// Mitsubishi GX Works2 project: 기말   PLC: Q02/Q02H

PROGRAM MAIN
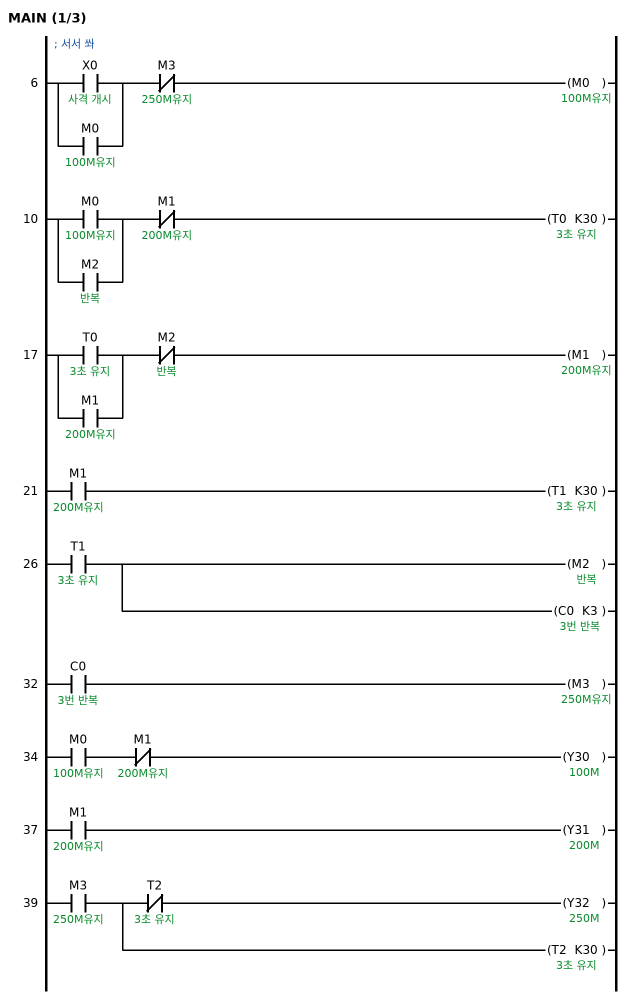
; 서서 쏴
6     LD      X0  ; 사격 개시
      OR      M0  ; 100M유지
      ANI     M3  ; 250M유지
      OUT     M0  ; 100M유지
10    LD      M0  ; 100M유지
      OR      M2  ; 반복
      ANI     M1  ; 200M유지
      OUT     T0 K30  ; 3초 유지
17    LD      T0  ; 3초 유지
      OR      M1  ; 200M유지
      ANI     M2  ; 반복
      OUT     M1  ; 200M유지
21    LD      M1  ; 200M유지
      OUT     T1 K30  ; 3초 유지
26    LD      T1  ; 3초 유지
      OUT     M2  ; 반복
      OUT     C0 K3  ; 3번 반복
32    LD      C0  ; 3번 반복
      OUT     M3  ; 250M유지
34    LD      M0  ; 100M유지
      ANI     M1  ; 200M유지
      OUT     Y30  ; 100M
37    LD      M1  ; 200M유지
      OUT     Y31  ; 200M
39    LD      M3  ; 250M유지
      MPS
      ANI     T2  ; 3초 유지
      OUT     Y32  ; 250M
      MPP
      OUT     T2 K30  ; 3초 유지
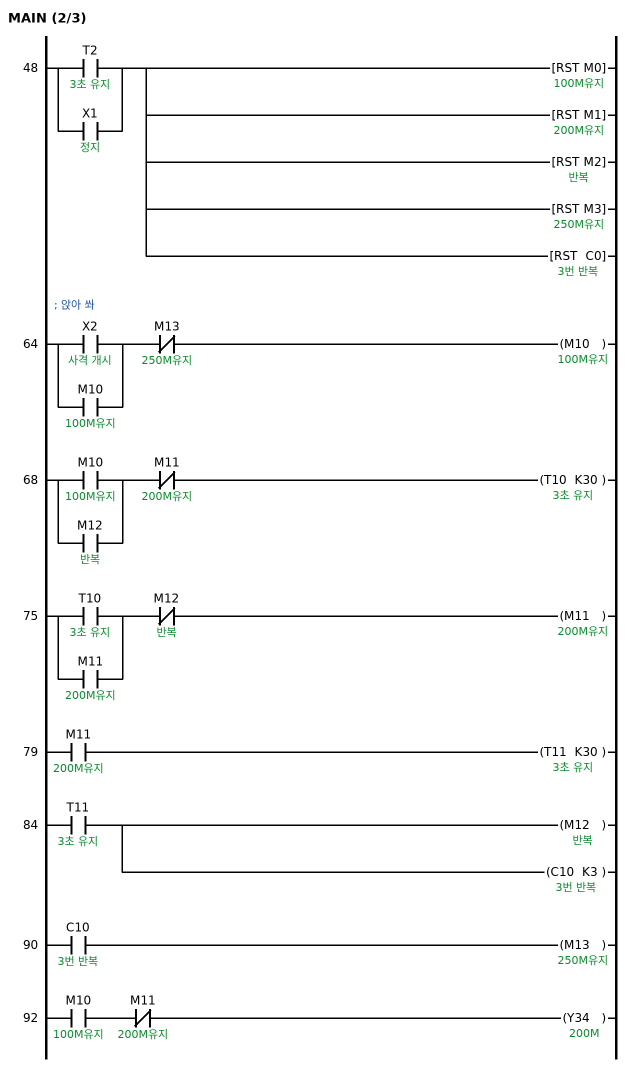
48    LD      T2  ; 3초 유지
      OR      X1  ; 정지
      RST     M0  ; 100M유지
      RST     M1  ; 200M유지
      RST     M2  ; 반복
      RST     M3  ; 250M유지
      RST     C0  ; 3번 반복
; 앉아 쏴
64    LD      X2  ; 사격 개시
      OR      M10  ; 100M유지
      ANI     M13  ; 250M유지
      OUT     M10  ; 100M유지
68    LD      M10  ; 100M유지
      OR      M12  ; 반복
      ANI     M11  ; 200M유지
      OUT     T10 K30  ; 3초 유지
75    LD      T10  ; 3초 유지
      OR      M11  ; 200M유지
      ANI     M12  ; 반복
      OUT     M11  ; 200M유지
79    LD      M11  ; 200M유지
      OUT     T11 K30  ; 3초 유지
84    LD      T11  ; 3초 유지
      OUT     M12  ; 반복
      OUT     C10 K3  ; 3번 반복
90    LD      C10  ; 3번 반복
      OUT     M13  ; 250M유지
92    LD      M10  ; 100M유지
      ANI     M11  ; 200M유지
      OUT     Y34  ; 200M
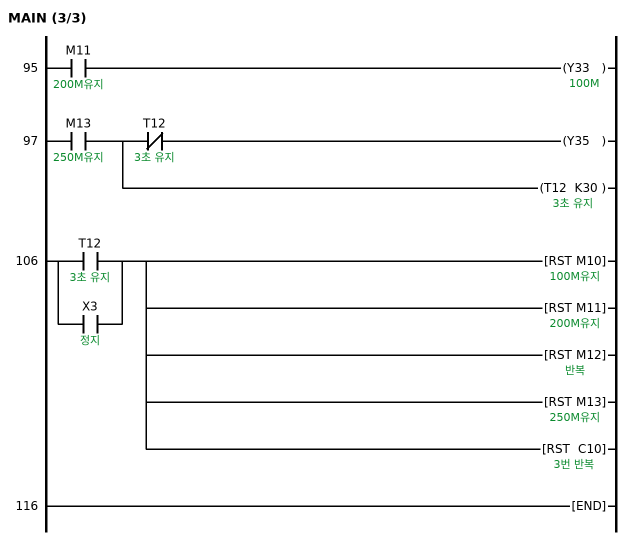
95    LD      M11  ; 200M유지
      OUT     Y33  ; 100M
97    LD      M13  ; 250M유지
      MPS
      ANI     T12  ; 3초 유지
      OUT     Y35
      MPP
      OUT     T12 K30  ; 3초 유지
106   LD      T12  ; 3초 유지
      OR      X3  ; 정지
      RST     M10  ; 100M유지
      RST     M11  ; 200M유지
      RST     M12  ; 반복
      RST     M13  ; 250M유지
      RST     C10  ; 3번 반복
116   END
END_PROGRAM
